// TwinCAT 3 PLC project PLC
// ProgramVersion: 3.1.4024.0
// libraries:
//   Tc2_EtherCAT, * (Beckhoff Automation GmbH)
//   Tc2_Standard, * (Beckhoff Automation GmbH)
//   Tc2_System, * (Beckhoff Automation GmbH)
//   Tc3_Module, * (Beckhoff Automation GmbH)
// project tree:
//   DUTs/ E_EP7402_CoE_Motor.TcDUT, E_EP7402_CoE_Controller.TcDUT, E_SynchronInfoData.TcDUT, ST_CoE_Parameter.TcDUT, ST_EP7402_CoE_Motor.TcDUT, ST_EP7402_CoE_Controller.TcDUT, ST_EP7402_CoE_Parameter.TcDUT, ST_EP7402_CoE_SynchronInfoData.TcDUT
//   GVLs/ GVL.TcGVL
//   / PlcTask.TcTTO
//   POUs/CoE_Access/ FB_EP7402_AutoRequestSteps.TcPOU, FB_EP7402_ReadCoEParameter.TcPOU, FB_EP7402_Scan_Motor.TcPOU, FB_EP7402_WriteCoEParameter.TcPOU
//   POUs/ MAIN.TcPOU
// real-time tasks:
//   TASK PlcTask: cycle T#2ms, priority 20, ADS port 350
// I/O:
//   DEVICE Device 3 (EtherCAT), AmsNetId 5.32.108.108.4.1
//     Box 1 (EP7402-0057) [EP7402-0057 2 Ch. BLDC Motor, 24VDC, 8x digital In/Output, B23 ENP 5G4, 1x EtherCAT junction]
// variable links:
//   PLC/PLC Instance <-> Device 3 (EtherCAT)/Box 1 (EP7402-0057)
//     PlcTask Inputs/MAIN.nEP7402Addr <-> InfoData/AdsAddr/port
//     PlcTask Inputs/MAIN.sNetId <-> InfoData/AdsAddr/netId
//     PlcTask Inputs/MAIN.stEP7402_PDOs.MDP5001_100_200_705_Input/MDP5001_100_200_705_STM_Inputs_Device_Device_Diag <-> STM Inputs Device/Device Diag
//     PlcTask Inputs/MAIN.stEP7402_PDOs.MDP5001_100_200_705_Input/MDP5001_100_DI_Inputs_Control_input_{1..4} <-> DI Inputs/Control input {1..4}  (4 links)
//     PlcTask Inputs/MAIN.stEP7402_PDOs.MDP5001_100_200_705_Input/MDP5001_100_DI_Inputs_Input_{1..4} <-> DI Inputs/Input {1..4}  (4 links)
//     PlcTask Inputs/MAIN.stEP7402_PDOs.MDP5001_100_200_705_Input/MDP5001_705_STM_Status_Channel_1_Status <-> STM Status Channel 1/Status
//     PlcTask Inputs/MAIN.stEP7402_PDOs.MDP5001_100_200_705_Input/MDP5001_705_STM_Status_Channel_2_Status <-> STM Status Channel 2/Status
//     PlcTask Inputs/MAIN.stEP7402_PDOs.MDP5001_100_200_705_Input/MDP5001_705_STM_Synchron_info_data_Channel_1_Info_data_1 <-> STM Synchron info data Channel 1/Info data 1
//     PlcTask Inputs/MAIN.stEP7402_PDOs.MDP5001_100_200_705_Input/MDP5001_705_STM_Synchron_info_data_Channel_1_Info_data_2 <-> STM Synchron info data Channel 1/Info data 2
//     PlcTask Inputs/MAIN.stEP7402_PDOs.MDP5001_100_200_705_Input/MDP5001_705_STM_Synchron_info_data_Channel_1_Info_data_3 <-> STM Synchron info data Channel 1/Info data 3
//     PlcTask Inputs/MAIN.stEP7402_PDOs.MDP5001_100_200_705_Input/MDP5001_705_STM_Synchron_info_data_Channel_2_Info_data_1 <-> STM Synchron info data Channel 2/Info data 1
//     PlcTask Inputs/MAIN.stEP7402_PDOs.MDP5001_100_200_705_Input/MDP5001_705_STM_Synchron_info_data_Channel_2_Info_data_2 <-> STM Synchron info data Channel 2/Info data 2
//     PlcTask Inputs/MAIN.stEP7402_PDOs.MDP5001_100_200_705_Input/MDP5001_705_STM_Synchron_info_data_Channel_2_Info_data_3 <-> STM Synchron info data Channel 2/Info data 3
//     PlcTask Outputs/MAIN.stEP7402_PDOs.MDP5001_100_200_705_Output/MDP5001_200_DO_Outputs_Control_output_{1..4} <-> DO Outputs/Control output {1..4}  (4 links)
//     PlcTask Outputs/MAIN.stEP7402_PDOs.MDP5001_100_200_705_Output/MDP5001_200_DO_Outputs_Output_{1..4} <-> DO Outputs/Output {1..4}  (4 links)
//     PlcTask Outputs/MAIN.stEP7402_PDOs.MDP5001_100_200_705_Output/MDP5001_705_STM_Control_Channel_1_Control <-> STM Control Channel 1/Control
//     PlcTask Outputs/MAIN.stEP7402_PDOs.MDP5001_100_200_705_Output/MDP5001_705_STM_Control_Channel_2_Control <-> STM Control Channel 2/Control
//     PlcTask Outputs/MAIN.stEP7402_PDOs.MDP5001_100_200_705_Output/MDP5001_705_STM_Target_Velocity_Channel_1_Accelleration <-> STM Target Velocity Channel 1/Accelleration
//     PlcTask Outputs/MAIN.stEP7402_PDOs.MDP5001_100_200_705_Output/MDP5001_705_STM_Target_Velocity_Channel_2_Accelleration <-> STM Target Velocity Channel 2/Accelleration
//     PlcTask Outputs/MAIN.stEP7402_PDOs.MDP5001_100_200_705_Output/MDP5001_705_STM_Target_Velocity_Channel_1_Decceleration <-> STM Target Velocity Channel 1/Decceleration
//     PlcTask Outputs/MAIN.stEP7402_PDOs.MDP5001_100_200_705_Output/MDP5001_705_STM_Target_Velocity_Channel_2_Decceleration <-> STM Target Velocity Channel 2/Decceleration
//     PlcTask Outputs/MAIN.stEP7402_PDOs.MDP5001_100_200_705_Output/MDP5001_705_STM_Target_Velocity_Channel_1_Velocity <-> STM Target Velocity Channel 1/Velocity
//     PlcTask Outputs/MAIN.stEP7402_PDOs.MDP5001_100_200_705_Output/MDP5001_705_STM_Target_Velocity_Channel_2_Velocity <-> STM Target Velocity Channel 2/Velocity

CONFIGURATION PLC
    RESOURCE PLC ON TwinCAT3
        TASK PlcTask(INTERVAL := T#2ms, PRIORITY := 20);
        PROGRAM MAIN WITH PlcTask : MAIN;
    END_RESOURCE
END_CONFIGURATION

// ---- DUTs/E_EP7402_CoE_Motor.TcDUT
{attribute 'qualified_only'}
{attribute 'strict'}
TYPE E_EP7402_CoE_Motor :
(
	Peak_Current:=1,
	Rated_Current:=2,
	Rated_Voltage:=3,
	Phase_To_Phase_Resistance:=4,
	Start_Velocity:=5,
	Mechanical_To_Electrical_Ratio:=6,
	Rated_Velocity:=7,
	I2T_Warn_Level:=8,
	I2T_Error_Level:=9,
	Motor_Thermal_Time_Constant:=10
);
END_TYPE

// ---- DUTs/E_EP7402_CoE_Controller.TcDUT
{attribute 'qualified_only'}
{attribute 'strict'}
TYPE E_EP7402_CoE_Controller :
(
	Disable_Motor_Diagnosis:=1,
	Disable_I2T_Current_Limiting:=2,
	Velocity_Loop_Integral_Time:=3,
	Velocity_Loop_Proportional_Gain:=4,
	Velocity_Feed_Forward_Gain:=5,
	Sensorless_Offset_Scaling:=6,
	Align_Duration:=7,
	Rampup_Duration:=8,
	Rampup_Velocity:=9,	
	Rampup_Needed_Switchover_Events:=10,
	Commutation_Threshold:=11,
	Current_Loop_Proportional_Gain:=12,
	Current_Loop_Integral_Time:=13,
	Restart_After_Error_Number_Of_Repetition:=14,
	Restart_After_Error_Delay:=15
);
END_TYPE

// ---- DUTs/E_SynchronInfoData.TcDUT
{attribute 'qualified_only'}
TYPE E_SynchronInfoData :
(
	Motor_velocity 				:= 7,
	Motor_velocity_filtered 	:= 8,
	Motor_I2T_load 				:= 11,
	Amplifier_I2T_load 			:= 12,
	Motor_dc_current 			:= 13,
	Motor_dc_current_filtered 	:= 14,
	Motor_back_emf 				:= 17,
	Motor_restart_counter 		:= 18,
	Internal_temperature 		:= 101,
	Motor_supply_voltage 		:= 104,
	none
)USINT:=none;
END_TYPE

// ---- DUTs/ST_CoE_Parameter.TcDUT
TYPE ST_CoE_Parameter :
STRUCT
	sSubIndex		: STRING;	// Number of Index:Subindex
	sDescription	: STRING;	// Description of CoE Parameter
	nValue			: UDINT;	// Set Value to change CoE Parameter 
	nReadValue		: UDINT;	// Actual Value of Parameterread from terminal
	sValueRange		: STRING;	// Description of the range of the parameter 
END_STRUCT
END_TYPE

// ---- DUTs/ST_EP7402_CoE_Motor.TcDUT
 {attribute 'pack_mode' := '0'}
 // Represents data struct of COE Index 8020/8030 --> can be determined in esi
TYPE ST_EP7402_CoE_Motor :
STRUCT
	Sub_Index_res_0: ARRAY [1..2] OF BYTE;
	Sub_Index_001: UINT;
	Sub_Index_002: UINT;
	Sub_Index_003: UINT;
	Sub_Index_004: UINT;
	Sub_Index_res_1: ARRAY [1..8] OF BYTE;
	Sub_Index_009: UINT;
	Sub_Index_res_2: ARRAY [1..8] OF BYTE;	
	Sub_Index_019: UINT;
	Sub_Index_020: UINT;
	Sub_Index_res_3: ARRAY [1..2] OF BYTE;	
	Sub_Index_022: USINT;
	Sub_Index_024: USINT;
	Sub_Index_025: UINT;
	Sub_Index_res_4: ARRAY [1..2] OF BYTE;	
END_STRUCT
END_TYPE

// ---- DUTs/ST_EP7402_CoE_Controller.TcDUT
 {attribute 'pack_mode' := '0'}
 // Represents data struct of COE Index 8023/8033 --> can be determined in esi
TYPE ST_EP7402_CoE_Controller :
STRUCT
	Bit_Reserved_001 :BIT;
	Bit_Reserved_002 :BIT;
	Bit_Reserved_003 :BIT;
	Bit_Reserved_004 :BIT;
	Bit_Reserved_005 :BIT;
	Bit_Reserved_006 :BIT;
	Bit_Reserved_007 :BIT;
	Bit_Reserved_008 :BIT;
	Bit_Reserved_009 :BIT;
	Bit_Reserved_010 :BIT;
	Bit_Reserved_011 :BIT;
	Bit_Reserved_012 :BIT;
	Bit_Reserved_013 :BIT;
	Bit_Reserved_014 :BIT;
	Bit_Reserved_015 :BIT;
	Bit_Reserved_016 :BIT;
	Bit_Reserved_017 :BIT;
	Sub_Index_002: BIT;
	Sub_Index_003: BIT;
	Sub_Index_004: BIT;
	Bit_Reserved_021 :BIT;
	Bit_Reserved_022 :BIT;
	Bit_Reserved_023 :BIT;
	Bit_Reserved_024 :BIT;
	Bit_Reserved_025 :BIT;
	Bit_Reserved_026 :BIT;
	Bit_Reserved_027 :BIT;
	Bit_Reserved_028 :BIT;
	Bit_Reserved_029 :BIT;
	Bit_Reserved_030 :BIT;
	Bit_Reserved_031 :BIT;
	Bit_Reserved_032 :BIT;
	Sub_Index_017: UDINT;
	Sub_Index_018: UDINT;
	Sub_Index_019: USINT;
	Sub_Index_020: SINT;
	Sub_Index_021: UINT;
	Byte_Reserved_001 :ARRAY[1..2] OF BYTE;
	Sub_Index_024: UINT;
	Sub_Index_025: UINT;
	Sub_Index_033: UINT;
	Sub_Index_034: UINT;
	Sub_Index_035: UINT;
	Sub_Index_036: UINT;
	Sub_Index_037: UINT;
	Sub_Index_038: UINT;
END_STRUCT
END_TYPE

// ---- DUTs/ST_EP7402_CoE_Parameter.TcDUT
TYPE ST_EP7402_CoE_Parameter :
STRUCT
	astCoE_Parameter_Motor				: ARRAY[1..2] OF ARRAY [1..gvl.cnNumberOfCoeParameter_Motor] OF ST_CoE_Parameter :=
	[[
		(sSubIndex:='8020:01',	sDescription:='Peak current[mA]'					,nValue:=0,nReadValue:=0, sValueRange:='<5000'),
		(sSubIndex:='8020:02',	sDescription:='Rated current[mA]'					,nValue:=0,nReadValue:=0, sValueRange:='<3500'),
		(sSubIndex:='8020:03',	sDescription:='Rated Voltage [0.01 V]'				,nValue:=0,nReadValue:=0, sValueRange:='<2400'),
		(sSubIndex:='8020:04',	sDescription:='Phase to phase resistance [0.01 Ω]'	,nValue:=0,nReadValue:=0, sValueRange:='-'),
		(sSubIndex:='8020:09',	sDescription:='Start velocity [°/s]'				,nValue:=0,nReadValue:=0, sValueRange:='-'),
		(sSubIndex:='8020:13',	sDescription:='Mechanical to electrical ratio'		,nValue:=0,nReadValue:=0, sValueRange:='-'),
		(sSubIndex:='8020:14',	sDescription:='Rated velocity [°/s]'				,nValue:=0,nReadValue:=0, sValueRange:='-'),
		(sSubIndex:='8020:16',	sDescription:='I2T warn level [%]'					,nValue:=0,nReadValue:=0, sValueRange:='-'),
		(sSubIndex:='8020:18',	sDescription:='I2T error level [%]'					,nValue:=0,nReadValue:=0, sValueRange:='-'),
		(sSubIndex:='8020:19',	sDescription:='Motor thermal time constant [0.1s]'	,nValue:=0,nReadValue:=0, sValueRange:='-')
	],
	[
		(sSubIndex:='8030:01',	sDescription:='Peak current[mA]'					,nValue:=0,nReadValue:=0, sValueRange:='<5000'),
		(sSubIndex:='8030:02',	sDescription:='Rated current[mA]'					,nValue:=0,nReadValue:=0, sValueRange:='<3500'),
		(sSubIndex:='8030:03',	sDescription:='Rated Voltage [0.01 V]'				,nValue:=0,nReadValue:=0, sValueRange:='<2400'),
		(sSubIndex:='8030:04',	sDescription:='Phase to phase resistance [0.01 Ω]'	,nValue:=0,nReadValue:=0, sValueRange:='-'),
		(sSubIndex:='8030:09',	sDescription:='Start velocity [°/s]'				,nValue:=0,nReadValue:=0, sValueRange:='-'),
		(sSubIndex:='8030:13',	sDescription:='Mechanical to electrical ratio'		,nValue:=0,nReadValue:=0, sValueRange:='-'),
		(sSubIndex:='8030:14',	sDescription:='Rated velocity [°/s]'				,nValue:=0,nReadValue:=0, sValueRange:='-'),
		(sSubIndex:='8030:16',	sDescription:='I2T warn level [%]'					,nValue:=0,nReadValue:=0, sValueRange:='-'),
		(sSubIndex:='8030:18',	sDescription:='I2T error level [%]'					,nValue:=0,nReadValue:=0, sValueRange:='-'),
		(sSubIndex:='8030:19',	sDescription:='Motor thermal time constant [0.1s]'	,nValue:=0,nReadValue:=0, sValueRange:='-')
	]];
	
	astCoE_Parameter_Controller			: ARRAY[1..2] OF ARRAY [1..gvl.cnNumberOfCoeParameter_Controller] OF ST_CoE_Parameter :=
		[[
			(sSubIndex:='8023:03',	sDescription:='Disable motor diagnosis'						,nValue:=0,nReadValue:=0, sValueRange:='0/1'),
			(sSubIndex:='8023:04',	sDescription:='Disable I2T current limiting'				,nValue:=0,nReadValue:=0, sValueRange:='0/1'),
			(sSubIndex:='8023:11',	sDescription:='Velocity loop integral time [0.1ms]'			,nValue:=0,nReadValue:=0, sValueRange:='-'),
            (sSubIndex:='8023:12',	sDescription:='Velocity loop proportional gain [uV/(°/s)]'	,nValue:=0,nReadValue:=0, sValueRange:='-'),
            (sSubIndex:='8023:13',	sDescription:='Velocity feed forward'						,nValue:=0,nReadValue:=0, sValueRange:='-'),
            (sSubIndex:='8023:14',	sDescription:='Sensorless offset scaling {%]'				,nValue:=0,nReadValue:=0, sValueRange:='-'),
            (sSubIndex:='8023:15',	sDescription:='Align duration [ms]'							,nValue:=0,nReadValue:=0, sValueRange:='-'),
            (sSubIndex:='8023:18',	sDescription:='Rampup duration [ms]'						,nValue:=0,nReadValue:=0, sValueRange:='-'),
            (sSubIndex:='8023:19',	sDescription:='Rampup velocity [°/s]'						,nValue:=0,nReadValue:=0, sValueRange:='-'),
            (sSubIndex:='8023:21',	sDescription:='Rampup needed switchover events'				,nValue:=0,nReadValue:=0, sValueRange:='-'),
            (sSubIndex:='8023:22',	sDescription:='Commutation Threshold'						,nValue:=0,nReadValue:=0, sValueRange:='-'),
            (sSubIndex:='8023:23',	sDescription:='Current loop proportional gain [0.1V/A]'		,nValue:=0,nReadValue:=0, sValueRange:='-'),
            (sSubIndex:='8023:24',	sDescription:='Current Loop integral time [0.1ms]'			,nValue:=0,nReadValue:=0, sValueRange:='-'),
            (sSubIndex:='8023:25',	sDescription:='Restart after error number of repetition'	,nValue:=0,nReadValue:=0, sValueRange:='-'),
            (sSubIndex:='8023:26',	sDescription:='Restart after error delay [ms]'					,nValue:=0,nReadValue:=0, sValueRange:='-')
		],
		[
			(sSubIndex:='8033:03',	sDescription:='Disable motor diagnosis'						,nValue:=0,nReadValue:=0, sValueRange:='0/1'),
			(sSubIndex:='8033:04',	sDescription:='Disable I2T current limiting'				,nValue:=0,nReadValue:=0, sValueRange:='0/1'),
			(sSubIndex:='8033:11',	sDescription:='Velocity loop integral time [0.1ms]'			,nValue:=0,nReadValue:=0, sValueRange:='-'),
            (sSubIndex:='8033:12',	sDescription:='Velocity loop proportional gain [uV/(°/s)]'	,nValue:=0,nReadValue:=0, sValueRange:='-'),
            (sSubIndex:='8033:13',	sDescription:='Velocity feed forward'						,nValue:=0,nReadValue:=0, sValueRange:='-'),
            (sSubIndex:='8033:14',	sDescription:='Sensorless offset scaling {%]'				,nValue:=0,nReadValue:=0, sValueRange:='-'),
            (sSubIndex:='8033:15',	sDescription:='Align duration [ms]'							,nValue:=0,nReadValue:=0, sValueRange:='-'),
            (sSubIndex:='8033:18',	sDescription:='Rampup duration [ms]'						,nValue:=0,nReadValue:=0, sValueRange:='-'),
            (sSubIndex:='8033:19',	sDescription:='Rampup velocity [°/s]'						,nValue:=0,nReadValue:=0, sValueRange:='-'),
            (sSubIndex:='8033:21',	sDescription:='Rampup needed switchover events'				,nValue:=0,nReadValue:=0, sValueRange:='-'),
            (sSubIndex:='8033:22',	sDescription:='Commutation Threshold'						,nValue:=0,nReadValue:=0, sValueRange:='-'),
            (sSubIndex:='8033:23',	sDescription:='Current loop proportional gain [0.1V/A]'		,nValue:=0,nReadValue:=0, sValueRange:='-'),
            (sSubIndex:='8033:24',	sDescription:='Current Loop integral time [0.1ms]'		   	,nValue:=0,nReadValue:=0, sValueRange:='-'),
            (sSubIndex:='8033:25',	sDescription:='Restart after error number of repetition'	,nValue:=0,nReadValue:=0, sValueRange:='-'),
            (sSubIndex:='8033:26',	sDescription:='Restart after error delay [ms]'				,nValue:=0,nReadValue:=0, sValueRange:='-')
		]];
		astCoE_Parameter_SynchronInfoData	: ARRAY [1..2] OF ARRAY [1..3] OF E_SynchronInfoData;
END_STRUCT 
END_TYPE

// ---- DUTs/ST_EP7402_CoE_SynchronInfoData.TcDUT
 {attribute 'pack_mode' := '0'}
// Represents data struct of COE Index 8022/8032 --> can be determined in esi
TYPE ST_EP7402_CoE_SynchronInfoData :
STRUCT
	aSub_Index_res_000 : ARRAY [1..4] OF BYTE;
	nInfoData1 : USINT;
	nInfoData2 : USINT;
	aSub_Index_res_001 : ARRAY [1..6] OF BYTE;
	nInfoData3 : USINT;
	aSub_Index_res_002 : ARRAY [1..3] OF BYTE;	
END_STRUCT
END_TYPE

// ---- GVLs/GVL.TcGVL
{attribute 'qualified_only'}
VAR_GLOBAL CONSTANT
	cnNumberOfCoeParameter_Motor:USINT:=10;
	cnNumberOfCoeParameter_Controller:USINT:=15;
	cnSubIndex_ResetDeliveryStatus: BYTE:=16#1;
	cnIndex_ResetDeliveryStatus: WORD:=16#1011;
	cnResetParameter : UDINT:= 1684107116;
END_VAR

// ---- POUs/MAIN.TcPOU
PROGRAM MAIN
VAR
	// Variables to link with HW
	sNetId			AT%I*	: T_AmsNetIdArr;				// link with PDO: EP7402 -->InfoData --> AdsAddr.netId
	nEP7402Addr		AT%I*	: UINT := 1001;					// link with PDO: EP7402 -->InfoData --> AdsAddr.port
	stEP7402_PDOs			: MDP5001_100_200_705_F94A9C2E;	// Struct for simple Link with Box: EP7402 --> PLC --> Create PLC Data Type --> disable "Per Channel"
															// --> Link To PLC.. --> Select Struct this struct

	// Function blocks used for COE access 
	fbEP7402_ReadCoE 			: FB_EP7402_ReadCoEParameter; 	// Read Coe Settings for Motor Configuration: Index 8020/30 and 8023/33 of a box
	fbEP7402_WriteCoE 			: FB_EP7402_WriteCoEParameter;	// Write Coe Settings for Motor Configuration: Index 8020/30 and 8023/33 of a box
	fbEP7402_AutoRequestSteps	: FB_EP7402_AutoRequestSteps;	// Sending Request for single Motor steps. Needed to determine "Mechanical to electrical Ratio"
	fbEP7402_ScanMotor			: FB_EP7402_Scan_Motor;			// Sending Request to start Motor Scan. Needed to determine controller values.
	fbResetCoE_Parameter 		: FB_EcCoESdoWrite;				// Reset Box --> reset to delivery status
	
	// structs storing CoE-Parameters
	stLast_EP7402_CoE_Parameter : ST_EP7402_CoE_Parameter;		// Struct with Coe Paramters in last PLC Cycle --> needed for getting changes
	st_EP7402_CoE_Parameter 	: ST_EP7402_CoE_Parameter;		// Struct containing all current CoE Data (also inputs from HMI)
	
	fbCoeWriteFinished			: f_trig;
	fbReadFinished				: f_trig;
	bReadCoE					: BOOL;
	bMotorChannel_1_Selected	: BOOL:=True;
	nIndex						: UINT;	
	nResetParameter 			: UDINT;
	bInit						: BOOL;
END_VAR

GetEvents();
Init();

// Reset Box to delivery state (can be triggered from HMI)
fbResetCoE_Parameter(	sNetID:=F_CreateAmsNetId(sNetId),
						nSlaveAddr:=nEP7402Addr, 
						nSubIndex := gvl.cnSubIndex_ResetDeliveryStatus, 
						nIndex := gvl.cnIndex_ResetDeliveryStatus,	
						pSrcBuf := ADR(gvl.cnResetParameter),
						cbBufLen := SIZEOF(gvl.cnResetParameter),
						bExecute := fbResetCoE_Parameter.bExecute
						);

// special configuration functions requested via CoE (can be triggered from HMI)
	//Request single Motor Steps
	fbEP7402_AutoRequestSteps(bEnable:=fbEP7402_AutoRequestSteps.bEnable, bMotorChannel_1:=bMotorChannel_1_Selected,sNetID:=F_CreateAmsNetId(sNetId),nSlaveAddr:=nEP7402Addr);
	//Request Motor Scan
	fbEP7402_ScanMotor(bExecute:=fbEP7402_ScanMotor.bExecute, bMotorChannel_1:=bMotorChannel_1_Selected,sNetID:=F_CreateAmsNetId(sNetId),nSlaveAddr:=nEP7402Addr);

ACTION GetEvents:


// A Coe Write has finished --> Read is necessary
fbCoeWriteFinished(clk:=fbEP7402_WriteCoE.bBusy OR fbResetCoE_Parameter.bBusy OR fbEP7402_ScanMotor.bBusy);

// Read in CoE Parameters of Box
fbEP7402_ReadCoE(bExecute:=fbCoeWriteFinished.q OR fbEP7402_ReadCoE.bExecute AND NOT fbEP7402_WriteCoE.bBusy , stEP7402_CoE_Parameter  :=st_EP7402_CoE_Parameter);
// A Coe Read is finished
fbReadFinished(clk:=fbEP7402_ReadCoE.bBusy );
IF fbReadFinished.Q THEN
	fbEP7402_ReadCoE.bExecute:=false;
	initCoEValues();
END_IF

// Write Coe Parameters if set parameters have been changed (HMI)
fbEP7402_WriteCoE(bExecute:=FALSE, stEP7402_CoE_Parameter  :=st_EP7402_CoE_Parameter);
IF memcmp(ADR(stLast_EP7402_CoE_Parameter),ADR(st_EP7402_CoE_Parameter),SIZEOF(st_EP7402_CoE_Parameter))<>0 AND NOT fbEP7402_ReadCoE.bBusy THEN 
	fbEP7402_WriteCoE(bExecute:=TRUE, sNetID:=F_CreateAmsNetId(sNetId),nSlaveAddr:=nEP7402Addr, stEP7402_CoE_Parameter  :=st_EP7402_CoE_Parameter);
	stLast_EP7402_CoE_Parameter:=st_EP7402_CoE_Parameter;
END_IF
END_ACTION

ACTION Init:
IF NOT bInit THEN
	fbEP7402_ReadCoE(bExecute:=NOT fbEP7402_ReadCoE.bBusy,sNetID:=F_CreateAmsNetId(sNetId),nSlaveAddr:=nEP7402Addr, stEP7402_CoE_Parameter  :=st_EP7402_CoE_Parameter);
	IF NOT fbEP7402_ReadCoE.bBusy THEN
		bInit:=TRUE;
		initCoEValues();
	END_IF
END_IF
END_ACTION

ACTION InitCoEValues:
FOR nIndex:= 1 TO gvl.cnNumberOfCoeParameter_Motor DO
	st_EP7402_CoE_Parameter.astCoE_Parameter_Motor[1][nIndex].nValue:=st_EP7402_CoE_Parameter.astCoE_Parameter_Motor[1][nIndex].nReadValue;
	st_EP7402_CoE_Parameter.astCoE_Parameter_Motor[2][nIndex].nValue:=st_EP7402_CoE_Parameter.astCoE_Parameter_Motor[2][nIndex].nReadValue;
END_FOR
FOR nIndex:= 1 TO gvl.cnNumberOfCoeParameter_Controller DO
	st_EP7402_CoE_Parameter.astCoE_Parameter_Controller[1][nIndex].nValue:=st_EP7402_CoE_Parameter.astCoE_Parameter_Controller[1][nIndex].nReadValue;
	st_EP7402_CoE_Parameter.astCoE_Parameter_Controller[2][nIndex].nValue:=st_EP7402_CoE_Parameter.astCoE_Parameter_Controller[2][nIndex].nReadValue;
END_FOR
stLast_EP7402_CoE_Parameter:=st_EP7402_CoE_Parameter;
END_ACTION

END_PROGRAM

// ---- POUs/CoE_Access/FB_EP7402_ReadCoEParameter.TcPOU

FUNCTION_BLOCK FB_EP7402_ReadCoEParameter
VAR_IN_OUT 
	stEP7402_CoE_Parameter	: ST_EP7402_CoE_Parameter;		
END_VAR
VAR_INPUT
	bExecute	: BOOL;
	sNetId 		: T_AmsNetID;
	nSlaveAddr	: UINT;
END_VAR
VAR_OUTPUT
	bBusy:BOOL;
	bError:BOOL;
	nErrId:UDINT;
END_VAR
VAR
	fbReadCoEParameterEx				:  FB_EcCoESdoReadEx;
	nParameter							:  UINT;
	nStep								: (init, StartRead_MotorParameter_1, Reading_MotorParameter_1, StartRead_ControllerParameter_1, Reading_ControllerParameter_1, StartRead_SynchronInfoData_1, Reading_SynchronInfoData_1,
											StartRead_MotorParameter_2, Reading_MotorParameter_2, StartRead_ControllerParameter_2, Reading_ControllerParameter_2, StartRead_SynchronInfoData_2, Reading_SynchronInfoData_2);
	stCoe_Read_Motor					: ST_EP7402_CoE_Motor;
	stCoe_Read_Controller				: ST_EP7402_CoE_Controller;
	stCoe_Read_SynchronInfoData			: ST_EP7402_CoE_SynchronInfoData;
	fbExecuteTrigger				 	: r_trig;
	nIndex: uint;
END_VAR

fbExecuteTrigger(clk:=bExecute);
IF fbExecuteTrigger.q THEN
	nStep:=StartRead_MotorParameter_1;
	bBusy:=TRUE;
END_IF

CASE nStep OF
	init:
		bBusy := FALSE;
		bError:=fbReadCoEParameterEx.bError;
		nErrId:=fbReadCoEParameterEx.nErrId;
	
	StartRead_MotorParameter_1:
		fbReadCoEParameterEx(bExecute:=FALSE);
		IF NOT fbReadCoEParameterEx.bBusy THEN
			fbReadCoEParameterEx(
				sNetId:= sNetId, 
				nSlaveAddr:= nSlaveAddr, 
				nIndex:= 16#8020, 
				pDstBuf:= ADR(stCoe_Read_Motor), 
				cbBufLen:= SIZEOF(stCoe_Read_Motor), 
				bExecute:= TRUE,
				bCompleteAccess:= TRUE);
			nStep:=	Reading_MotorParameter_1;
		END_IF

		
	Reading_MotorParameter_1:
		fbReadCoEParameterEx(bExecute:=FALSE);
		IF NOT fbReadCoEParameterEx.bBusy THEN
			IF fbReadCoEParameterEx.bError THEN
				nStep:= init;
			ELSE
				TransferBufferDataToStruct_Motor(nChannel:=1);
				nStep:= StartRead_ControllerParameter_1;
			END_IF
		END_IF
	
	StartRead_ControllerParameter_1:
		fbReadCoEParameterEx(bExecute:=FALSE);
		IF NOT fbReadCoEParameterEx.bBusy THEN
			fbReadCoEParameterEx(
				sNetId:= sNetId, 
				nSlaveAddr:= nSlaveAddr, 
				nIndex:= 16#8023, 
				pDstBuf:= ADR(stCoe_Read_Controller), 
				cbBufLen:= SIZEOF(stCoe_Read_Controller), 
				bExecute:= TRUE,
				bCompleteAccess:= TRUE);
			nStep:=	Reading_ControllerParameter_1;
		END_IF
		
	Reading_ControllerParameter_1:
		fbReadCoEParameterEx(bExecute:=FALSE);
		IF NOT fbReadCoEParameterEx.bBusy THEN
			IF fbReadCoEParameterEx.bError THEN
				nStep:= init;
			ELSE
				TransferBufferDataToStruct_Controller(nChannel:=1);
				nStep:= StartRead_SynchronInfoData_1;
			END_IF
		END_IF
		
	StartRead_SynchronInfoData_1:
		fbReadCoEParameterEx(bExecute:=FALSE);
			IF NOT fbReadCoEParameterEx.bBusy THEN
				fbReadCoEParameterEx(
					sNetId:= sNetId, 
					nSlaveAddr:= nSlaveAddr, 
					nIndex:= 16#8022, 
					pDstBuf:= ADR(stCoe_Read_SynchronInfoData), 
					cbBufLen:= SIZEOF(stCoe_Read_SynchronInfoData), 
					bExecute:= TRUE,
					bCompleteAccess:= TRUE);
				nStep:=	Reading_SynchronInfoData_1;
			END_IF
	
	Reading_SynchronInfoData_1:
		fbReadCoEParameterEx(bExecute:=FALSE);
			IF NOT fbReadCoEParameterEx.bBusy THEN
				IF fbReadCoEParameterEx.bError THEN
					nStep:= init;
				ELSE
					TransferBufferDataToStruct_SynchronInfoData(nChannel:=1);
					nStep:= StartRead_MotorParameter_2;
				END_IF
			END_IF
		
	StartRead_MotorParameter_2:
		fbReadCoEParameterEx(bExecute:=FALSE);
		IF NOT fbReadCoEParameterEx.bBusy THEN
			fbReadCoEParameterEx(
				sNetId:= sNetId, 
				nSlaveAddr:= nSlaveAddr, 
				nIndex:= 16#8030, 
				pDstBuf:= ADR(stCoe_Read_Motor), 
				cbBufLen:= SIZEOF(stCoe_Read_Motor), 
				bExecute:= TRUE,
				bCompleteAccess:= TRUE);
			nStep:=	Reading_MotorParameter_2;
		END_IF

		
	Reading_MotorParameter_2:
		fbReadCoEParameterEx(bExecute:=FALSE);
		IF NOT fbReadCoEParameterEx.bBusy THEN
			IF fbReadCoEParameterEx.bError THEN
				nStep:= init;
			ELSE
				TransferBufferDataToStruct_Motor(nChannel:=2);
				nStep:= StartRead_ControllerParameter_2;
			END_IF
		END_IF
	
	StartRead_ControllerParameter_2:
		fbReadCoEParameterEx(bExecute:=FALSE);
		IF NOT fbReadCoEParameterEx.bBusy THEN
			fbReadCoEParameterEx(
				sNetId:= sNetId, 
				nSlaveAddr:= nSlaveAddr, 
				nIndex:= 16#8033, 
				pDstBuf:= ADR(stCoe_Read_Controller), 
				cbBufLen:= SIZEOF(stCoe_Read_Controller), 
				bExecute:= TRUE,
				bCompleteAccess:= TRUE);
			nStep:=	Reading_ControllerParameter_2;
		END_IF
		
	Reading_ControllerParameter_2:
		fbReadCoEParameterEx(bExecute:=FALSE);
		IF NOT fbReadCoEParameterEx.bBusy THEN
			IF fbReadCoEParameterEx.bError THEN
				nStep:= init;
			ELSE 
				TransferBufferDataToStruct_Controller(nChannel:=2);
				nStep:= StartRead_SynchronInfoData_2;
			END_IF
		END_IF
		
	StartRead_SynchronInfoData_2:
		fbReadCoEParameterEx(bExecute:=FALSE);
		IF NOT fbReadCoEParameterEx.bBusy THEN
			fbReadCoEParameterEx(
				sNetId:= sNetId, 
				nSlaveAddr:= nSlaveAddr, 
				nIndex:= 16#8032, 
				pDstBuf:= ADR(stCoe_Read_SynchronInfoData), 
				cbBufLen:= SIZEOF(stCoe_Read_SynchronInfoData), 
				bExecute:= TRUE,
				bCompleteAccess:= TRUE);
			nStep:=	Reading_SynchronInfoData_2;
		END_IF
		
	Reading_SynchronInfoData_2:
		fbReadCoEParameterEx(bExecute:=FALSE);
		IF NOT fbReadCoEParameterEx.bBusy THEN
			IF NOT fbReadCoEParameterEx.bError THEN
				TransferBufferDataToStruct_SynchronInfoData(nChannel:=2);
			END_IF
			nStep:= init;
		END_IF
		
END_CASE

METHOD TransferBufferDataToStruct_Controller
VAR_INPUT
	nChannel:USINT;
END_VAR
// The warning can be disabled here as the user is aware of the risk that the reference may not be valid by checking its validity
{warning disable C0371}

IF nChannel=1 OR nChannel=2  AND __ISVALIDREF(stEP7402_CoE_Parameter)THEN
	stEP7402_CoE_Parameter.astCoE_Parameter_Controller[nChannel][E_EP7402_CoE_Controller.Disable_Motor_Diagnosis].nReadValue:=TO_UDINT(stCoe_Read_Controller.Sub_Index_003);
	stEP7402_CoE_Parameter.astCoE_Parameter_Controller[nChannel][E_EP7402_CoE_Controller.Disable_I2T_Current_Limiting].nReadValue:=TO_UDINT(stCoe_Read_Controller.Sub_Index_004);
	stEP7402_CoE_Parameter.astCoE_Parameter_Controller[nChannel][E_EP7402_CoE_Controller.Velocity_Loop_Integral_Time].nReadValue:=TO_UDINT(stCoe_Read_Controller.Sub_Index_017);
	stEP7402_CoE_Parameter.astCoE_Parameter_Controller[nChannel][E_EP7402_CoE_Controller.Velocity_Loop_Proportional_Gain].nReadValue:=TO_UDINT(stCoe_Read_Controller.Sub_Index_018);
	stEP7402_CoE_Parameter.astCoE_Parameter_Controller[nChannel][E_EP7402_CoE_Controller.Velocity_Feed_Forward_Gain].nReadValue:=TO_UDINT(stCoe_Read_Controller.Sub_Index_019);
	stEP7402_CoE_Parameter.astCoE_Parameter_Controller[nChannel][E_EP7402_CoE_Controller.Sensorless_Offset_Scaling].nReadValue:=TO_UDINT(stCoe_Read_Controller.Sub_Index_020);
	stEP7402_CoE_Parameter.astCoE_Parameter_Controller[nChannel][E_EP7402_CoE_Controller.Align_Duration].nReadValue:=TO_UDINT(stCoe_Read_Controller.Sub_Index_021);
	stEP7402_CoE_Parameter.astCoE_Parameter_Controller[nChannel][E_EP7402_CoE_Controller.Rampup_Duration].nReadValue:=TO_UDINT(stCoe_Read_Controller.Sub_Index_024);
	stEP7402_CoE_Parameter.astCoE_Parameter_Controller[nChannel][E_EP7402_CoE_Controller.Rampup_Velocity].nReadValue:=TO_UDINT(stCoe_Read_Controller.Sub_Index_025);
	stEP7402_CoE_Parameter.astCoE_Parameter_Controller[nChannel][E_EP7402_CoE_Controller.Rampup_Needed_Switchover_Events].nReadValue:=TO_UDINT(stCoe_Read_Controller.Sub_Index_033);
	stEP7402_CoE_Parameter.astCoE_Parameter_Controller[nChannel][E_EP7402_CoE_Controller.Commutation_Threshold].nReadValue:=TO_UDINT(stCoe_Read_Controller.Sub_Index_034);
	stEP7402_CoE_Parameter.astCoE_Parameter_Controller[nChannel][E_EP7402_CoE_Controller.Current_Loop_Proportional_Gain].nReadValue:=TO_UDINT(stCoe_Read_Controller.Sub_Index_035);
	stEP7402_CoE_Parameter.astCoE_Parameter_Controller[nChannel][E_EP7402_CoE_Controller.Current_Loop_Integral_Time].nReadValue:=TO_UDINT(stCoe_Read_Controller.Sub_Index_036);
	stEP7402_CoE_Parameter.astCoE_Parameter_Controller[nChannel][E_EP7402_CoE_Controller.Restart_After_Error_Number_Of_Repetition].nReadValue:=TO_UDINT(stCoe_Read_Controller.Sub_Index_037);
	stEP7402_CoE_Parameter.astCoE_Parameter_Controller[nChannel][E_EP7402_CoE_Controller.Restart_After_Error_Delay].nReadValue:=TO_UDINT(stCoe_Read_Controller.Sub_Index_038);
END_IF
END_METHOD

METHOD TransferBufferDataToStruct_Motor
VAR_INPUT
	nChannel:USINT;
END_VAR
// The warning can be disabled here as the user is aware of the risk that the reference may not be valid by checking its validity
{warning disable C0371}

IF nChannel=1 OR nChannel=2 and __ISVALIDREF(stEP7402_CoE_Parameter) THEN
	stEP7402_CoE_Parameter.astCoE_Parameter_Motor[nChannel][E_EP7402_CoE_Motor.Peak_Current].nReadValue:=stCoe_Read_Motor.Sub_Index_001;
	stEP7402_CoE_Parameter.astCoE_Parameter_Motor[nChannel][E_EP7402_CoE_Motor.Rated_Current].nReadValue:=stCoe_Read_Motor.Sub_Index_002;
	stEP7402_CoE_Parameter.astCoE_Parameter_Motor[nChannel][E_EP7402_CoE_Motor.Rated_Voltage].nReadValue:=stCoe_Read_Motor.Sub_Index_003;
	stEP7402_CoE_Parameter.astCoE_Parameter_Motor[nChannel][E_EP7402_CoE_Motor.Phase_To_Phase_Resistance].nReadValue:=stCoe_Read_Motor.Sub_Index_004;
	stEP7402_CoE_Parameter.astCoE_Parameter_Motor[nChannel][E_EP7402_CoE_Motor.Start_Velocity].nReadValue:=stCoe_Read_Motor.Sub_Index_009;
	stEP7402_CoE_Parameter.astCoE_Parameter_Motor[nChannel][E_EP7402_CoE_Motor.Mechanical_To_Electrical_Ratio].nReadValue:=stCoe_Read_Motor.Sub_Index_019;
	stEP7402_CoE_Parameter.astCoE_Parameter_Motor[nChannel][E_EP7402_CoE_Motor.Rated_Velocity].nReadValue:=stCoe_Read_Motor.Sub_Index_020;
	stEP7402_CoE_Parameter.astCoE_Parameter_Motor[nChannel][E_EP7402_CoE_Motor.I2T_Warn_Level].nReadValue:=stCoe_Read_Motor.Sub_Index_022;
	stEP7402_CoE_Parameter.astCoE_Parameter_Motor[nChannel][E_EP7402_CoE_Motor.I2T_Error_Level].nReadValue:=stCoe_Read_Motor.Sub_Index_024;
	stEP7402_CoE_Parameter.astCoE_Parameter_Motor[nChannel][E_EP7402_CoE_Motor.Motor_Thermal_Time_Constant].nReadValue:=stCoe_Read_Motor.Sub_Index_025;
END_IF
END_METHOD

METHOD TransferBufferDataToStruct_SynchronInfoData
VAR_INPUT
	nChannel:USINT;
END_VAR
// The warning can be disabled here as the user is aware of the risk that the reference may not be valid by checking its validity
{warning disable C0371}

IF nChannel=1 OR nChannel=2 and __ISVALIDREF(stEP7402_CoE_Parameter) THEN
	stEP7402_CoE_Parameter.astCoE_Parameter_SynchronInfoData[nChannel][1]:=stCoe_Read_SynchronInfoData.nInfoData1;
	stEP7402_CoE_Parameter.astCoE_Parameter_SynchronInfoData[nChannel][2]:=stCoe_Read_SynchronInfoData.nInfoData2;
	stEP7402_CoE_Parameter.astCoE_Parameter_SynchronInfoData[nChannel][3]:=stCoe_Read_SynchronInfoData.nInfoData3;
END_IF
END_METHOD

END_FUNCTION_BLOCK

// ---- POUs/CoE_Access/FB_EP7402_WriteCoEParameter.TcPOU
FUNCTION_BLOCK FB_EP7402_WriteCoEParameter
VAR_IN_OUT 
	stEP7402_CoE_Parameter	: ST_EP7402_CoE_Parameter;		
END_VAR
VAR_INPUT
	bExecute	: BOOL;
	sNetId 		: T_AmsNetID;
	nSlaveAddr	: UINT;
END_VAR
VAR_OUTPUT
	bBusy:BOOL;
	bError:BOOL;
	nErrId:UDINT;
END_VAR
VAR
	fbWriteCoEParameterEx				:  FB_EcCoESdoWriteEx;
	nParameter							:  UINT;
	nStep								: (init, StartSend_MotorParameter_1, Sending_MotorParameter_1, StartSend_ControllerParameter_1, Sending_ControllerParameter_1, StartSend_SynchronInfoData_1, Sending_SynchronInfoData_1,
											StartSend_MotorParameter_2, Sending_MotorParameter_2, StartSend_ControllerParameter_2, Sending_ControllerParameter_2, StartSend_SynchronInfoData_2, Sending_SynchronInfoData_2);
	stCoe_Write_Motor					: ST_EP7402_CoE_Motor;
	stCoe_Write_Controller				: ST_EP7402_CoE_Controller;
	stCoe_Write_SynchronInfoData		: ST_EP7402_CoE_SynchronInfoData;
	fbExecuteTrigger				 	: r_trig;
	nIndex: uint;
END_VAR

fbExecuteTrigger(clk:=bExecute);
IF fbExecuteTrigger.q THEN
	nStep:=StartSend_MotorParameter_1;
	bBusy:=TRUE;
END_IF

CASE nStep OF
	init:
		bBusy := FALSE;
		bError:=fbWriteCoEParameterEx.bError;
		nErrId:=fbWriteCoEParameterEx.nErrId;
	
	StartSend_MotorParameter_1:
		fbWriteCoEParameterEx(bExecute:=FALSE);
		IF NOT fbWriteCoEParameterEx.bBusy THEN
			TransferStructDataToBuffer_Motor(nChannel:=1);
			fbWriteCoEParameterEx(
				sNetId:= sNetId, 
				nSlaveAddr:= nSlaveAddr, 
				nIndex:= 16#8020, 
				pSrcBuf:= ADR(stCoe_Write_Motor), 
				cbBufLen:= SIZEOF(stCoe_Write_Motor), 
				bExecute:= TRUE,
				bCompleteAccess:= TRUE);
			nStep:=	Sending_MotorParameter_1;
		END_IF

		
	Sending_MotorParameter_1:
		fbWriteCoEParameterEx(bExecute:=FALSE);
		IF NOT fbWriteCoEParameterEx.bBusy THEN
			IF fbWriteCoEParameterEx.bError THEN
				nStep:= init;
			ELSE
				nStep:= StartSend_ControllerParameter_1;
			END_IF
		END_IF
	
	StartSend_ControllerParameter_1:
		fbWriteCoEParameterEx(bExecute:=FALSE);
		IF NOT fbWriteCoEParameterEx.bBusy THEN
			TransferStructDataToBuffer_Controller(nChannel:=1);
			fbWriteCoEParameterEx(
				sNetId:= sNetId, 
				nSlaveAddr:= nSlaveAddr, 
				nIndex:= 16#8023, 
				pSrcBuf:= ADR(stCoe_Write_Controller), 
				cbBufLen:= SIZEOF(stCoe_Write_Controller), 
				bExecute:= TRUE,
				bCompleteAccess:= TRUE);
			nStep:=	Sending_ControllerParameter_1;
		END_IF
		
	Sending_ControllerParameter_1:
		fbWriteCoEParameterEx(bExecute:=FALSE);
		IF NOT fbWriteCoEParameterEx.bBusy THEN
			IF fbWriteCoEParameterEx.bError THEN
				nStep:= init;
			ELSE
				nStep:= StartSend_SynchronInfoData_1;
			END_IF
		END_IF
		
	StartSend_SynchronInfoData_1:		
		fbWriteCoEParameterEx(bExecute:=FALSE);
		IF NOT fbWriteCoEParameterEx.bBusy THEN
			TransferStructDataToBuffer_SynchronInfoData(nChannel:=1);
			fbWriteCoEParameterEx(
				sNetId:= sNetId, 
				nSlaveAddr:= nSlaveAddr, 
				nIndex:= 16#8022, 
				pSrcBuf:= ADR(stCoe_Write_SynchronInfoData), 
				cbBufLen:= SIZEOF(stCoe_Write_SynchronInfoData), 
				bExecute:= TRUE,
				bCompleteAccess:= TRUE);
			nStep:=	Sending_SynchronInfoData_1;
		END_IF
		
	Sending_SynchronInfoData_1:
		fbWriteCoEParameterEx(bExecute:=FALSE);
		IF NOT fbWriteCoEParameterEx.bBusy THEN
			IF fbWriteCoEParameterEx.bError THEN
				nStep:= init;
			ELSE
				nStep:= StartSend_MotorParameter_2;
			END_IF
		END_IF
		
	StartSend_MotorParameter_2:
		fbWriteCoEParameterEx(bExecute:=FALSE);
		IF NOT fbWriteCoEParameterEx.bBusy THEN						
			TransferStructDataToBuffer_Motor(nChannel:=2);
			fbWriteCoEParameterEx(
				sNetId:= sNetId, 
				nSlaveAddr:= nSlaveAddr, 
				nIndex:= 16#8030, 
				pSrcBuf:= ADR(stCoe_Write_Motor), 
				cbBufLen:= SIZEOF(stCoe_Write_Motor), 
				bExecute:= TRUE,
				bCompleteAccess:= TRUE);
			nStep:=	Sending_MotorParameter_2;
		END_IF
		
	Sending_MotorParameter_2:
		fbWriteCoEParameterEx(bExecute:=FALSE);
		IF NOT fbWriteCoEParameterEx.bBusy THEN
			IF fbWriteCoEParameterEx.bError THEN
				nStep:= init;
			ELSE
				nStep:= StartSend_ControllerParameter_2;
			END_IF
		END_IF
	
	StartSend_ControllerParameter_2:
		fbWriteCoEParameterEx(bExecute:=FALSE);
		IF NOT fbWriteCoEParameterEx.bBusy THEN					
			TransferStructDataToBuffer_Controller(nChannel:=2);
			fbWriteCoEParameterEx(
				sNetId:= sNetId, 
				nSlaveAddr:= nSlaveAddr, 
				nIndex:= 16#8033, 
				pSrcBuf:= ADR(stCoe_Write_Controller), 
				cbBufLen:= SIZEOF(stCoe_Write_Controller), 
				bExecute:= TRUE,
				bCompleteAccess:= TRUE);
			nStep:=	Sending_ControllerParameter_2;
		END_IF
		
	Sending_ControllerParameter_2:
		fbWriteCoEParameterEx(bExecute:=FALSE);
		IF NOT fbWriteCoEParameterEx.bBusy THEN
			IF fbWriteCoEParameterEx.bError THEN
				nStep:= init;
			ELSE
				nStep:= StartSend_SynchronInfoData_2;
			END_IF
		END_IF
		
	StartSend_SynchronInfoData_2:
		fbWriteCoEParameterEx(bExecute:=FALSE);
		IF NOT fbWriteCoEParameterEx.bBusy THEN
			TransferStructDataToBuffer_SynchronInfoData(nChannel:=2);
			fbWriteCoEParameterEx(
				sNetId:= sNetId, 
				nSlaveAddr:= nSlaveAddr, 
				nIndex:= 16#8032, 
				pSrcBuf:= ADR(stCoe_Write_SynchronInfoData), 
				cbBufLen:= SIZEOF(stCoe_Write_SynchronInfoData), 
				bExecute:= TRUE,
				bCompleteAccess:= TRUE);
			nStep :=	Sending_SynchronInfoData_2;
		END_IF
		
	Sending_SynchronInfoData_2:
		fbWriteCoEParameterEx(bExecute:=FALSE);
		IF NOT fbWriteCoEParameterEx.bBusy THEN
				nStep:= init;
		END_IF
		
END_CASE

METHOD TransferStructDataToBuffer_Controller
VAR_INPUT
	nChannel:USINT;
END_VAR
// The warning can be disabled here as the user is aware of the risk that the reference may not be valid by checking its validity
{warning disable C0371}
IF nChannel=1 OR nChannel=2 AND __ISVALIDREF(stEP7402_CoE_Parameter) THEN
	stCoe_Write_Controller.Sub_Index_003	:= stEP7402_CoE_Parameter.astCoE_Parameter_Controller[nChannel][E_EP7402_CoE_Controller.Disable_Motor_Diagnosis].nValue.0;            
	stCoe_Write_Controller.Sub_Index_004	:= stEP7402_CoE_Parameter.astCoE_Parameter_Controller[nChannel][E_EP7402_CoE_Controller.Disable_I2T_Current_Limiting].nValue.0;        
	stCoe_Write_Controller.Sub_Index_017	:= stEP7402_CoE_Parameter.astCoE_Parameter_Controller[nChannel][E_EP7402_CoE_Controller.Velocity_Loop_Integral_Time].nValue;         
	stCoe_Write_Controller.Sub_Index_018	:= stEP7402_CoE_Parameter.astCoE_Parameter_Controller[nChannel][E_EP7402_CoE_Controller.Velocity_Loop_Proportional_Gain].nValue;      
	stCoe_Write_Controller.Sub_Index_019	:= TO_USINT(stEP7402_CoE_Parameter.astCoE_Parameter_Controller[nChannel][E_EP7402_CoE_Controller.Velocity_Feed_Forward_Gain].nValue);          
	stCoe_Write_Controller.Sub_Index_020	:= TO_SINT(stEP7402_CoE_Parameter.astCoE_Parameter_Controller[nChannel][E_EP7402_CoE_Controller.Sensorless_Offset_Scaling].nValue);          
	stCoe_Write_Controller.Sub_Index_021	:= TO_UINT(stEP7402_CoE_Parameter.astCoE_Parameter_Controller[nChannel][E_EP7402_CoE_Controller.Align_Duration].nValue);                   
	stCoe_Write_Controller.Sub_Index_024	:= TO_UINT(stEP7402_CoE_Parameter.astCoE_Parameter_Controller[nChannel][E_EP7402_CoE_Controller.Rampup_Duration].nValue);                  
	stCoe_Write_Controller.Sub_Index_025	:= TO_UINT(stEP7402_CoE_Parameter.astCoE_Parameter_Controller[nChannel][E_EP7402_CoE_Controller.Rampup_Velocity].nValue);                  
	stCoe_Write_Controller.Sub_Index_033	:= TO_UINT(stEP7402_CoE_Parameter.astCoE_Parameter_Controller[nChannel][E_EP7402_CoE_Controller.Rampup_Needed_Switchover_Events].nValue);      
	stCoe_Write_Controller.Sub_Index_034	:= TO_UINT(stEP7402_CoE_Parameter.astCoE_Parameter_Controller[nChannel][E_EP7402_CoE_Controller.Commutation_Threshold].nValue);             
	stCoe_Write_Controller.Sub_Index_035	:= TO_UINT(stEP7402_CoE_Parameter.astCoE_Parameter_Controller[nChannel][E_EP7402_CoE_Controller.Current_Loop_Proportional_Gain].nValue);       
	stCoe_Write_Controller.Sub_Index_036	:= TO_UINT(stEP7402_CoE_Parameter.astCoE_Parameter_Controller[nChannel][E_EP7402_CoE_Controller.Current_Loop_Integral_Time].nValue);          
	stCoe_Write_Controller.Sub_Index_037	:= TO_UINT(stEP7402_CoE_Parameter.astCoE_Parameter_Controller[nChannel][E_EP7402_CoE_Controller.Restart_After_Error_Number_Of_Repetition].nValue);
	stCoe_Write_Controller.Sub_Index_038	:= TO_UINT(stEP7402_CoE_Parameter.astCoE_Parameter_Controller[nChannel][E_EP7402_CoE_Controller.Restart_After_Error_Delay].nValue);          
END_IF
END_METHOD

METHOD TransferStructDataToBuffer_Motor
VAR_INPUT
	nChannel:USINT;
END_VAR
// The warning can be disabled here as the user is aware of the risk that the reference may not be valid by checking its validity
{warning disable C0371}

IF nChannel=1 OR nChannel=2 AND __ISVALIDREF(stEP7402_CoE_Parameter) THEN
	stCoe_Write_Motor.Sub_Index_001	:= TO_UINT(stEP7402_CoE_Parameter.astCoE_Parameter_Motor[nChannel][E_EP7402_CoE_Motor.Peak_Current].nValue);
	stCoe_Write_Motor.Sub_Index_002	:= TO_UINT(stEP7402_CoE_Parameter.astCoE_Parameter_Motor[nChannel][E_EP7402_CoE_Motor.Rated_Current].nValue);
	stCoe_Write_Motor.Sub_Index_003	:= TO_UINT(stEP7402_CoE_Parameter.astCoE_Parameter_Motor[nChannel][E_EP7402_CoE_Motor.Rated_Voltage].nValue);
	stCoe_Write_Motor.Sub_Index_004	:= TO_UINT(stEP7402_CoE_Parameter.astCoE_Parameter_Motor[nChannel][E_EP7402_CoE_Motor.Phase_To_Phase_Resistance].nValue);
	stCoe_Write_Motor.Sub_Index_009	:= TO_UINT(stEP7402_CoE_Parameter.astCoE_Parameter_Motor[nChannel][E_EP7402_CoE_Motor.Start_Velocity].nValue);
	stCoe_Write_Motor.Sub_Index_019	:= TO_UINT(stEP7402_CoE_Parameter.astCoE_Parameter_Motor[nChannel][E_EP7402_CoE_Motor.Mechanical_To_Electrical_Ratio].nValue);
	stCoe_Write_Motor.Sub_Index_020	:= TO_UINT(stEP7402_CoE_Parameter.astCoE_Parameter_Motor[nChannel][E_EP7402_CoE_Motor.Rated_Velocity].nValue);
	stCoe_Write_Motor.Sub_Index_022	:= TO_USINT(stEP7402_CoE_Parameter.astCoE_Parameter_Motor[nChannel][E_EP7402_CoE_Motor.I2T_Warn_Level].nValue);
	stCoe_Write_Motor.Sub_Index_024	:= TO_USINT(stEP7402_CoE_Parameter.astCoE_Parameter_Motor[nChannel][E_EP7402_CoE_Motor.I2T_Error_Level].nValue);
	stCoe_Write_Motor.Sub_Index_025	:= TO_UINT(stEP7402_CoE_Parameter.astCoE_Parameter_Motor[nChannel][E_EP7402_CoE_Motor.Motor_Thermal_Time_Constant].nValue);
END_IF
END_METHOD

METHOD TransferStructDataToBuffer_SynchronInfoData
VAR_INPUT
	nChannel:USINT;
END_VAR
// The warning can be disabled here as the user is aware of the risk that the reference may not be valid by checking its validity
{warning disable C0371}

IF nChannel=1 OR nChannel=2 AND __ISVALIDREF(stEP7402_CoE_Parameter) THEN
	stCoe_Write_SynchronInfoData.nInfoData1	:= TO_USINT(stEP7402_CoE_Parameter.astCoE_Parameter_SynchronInfoData[nChannel][1]);
	stCoe_Write_SynchronInfoData.nInfoData2	:= TO_USINT(stEP7402_CoE_Parameter.astCoE_Parameter_SynchronInfoData[nChannel][2]);
	stCoe_Write_SynchronInfoData.nInfoData3	:= TO_USINT(stEP7402_CoE_Parameter.astCoE_Parameter_SynchronInfoData[nChannel][3]);
END_IF
END_METHOD

END_FUNCTION_BLOCK

// ---- POUs/CoE_Access/FB_EP7402_AutoRequestSteps.TcPOU
FUNCTION_BLOCK FB_EP7402_AutoRequestSteps
VAR CONSTANT
	cnValueChannel_1: UINT:=16#800A;
	cnValueChannel_2: UINT:=16#801A;
END_VAR
VAR_INPUT
	bEnable:BOOL;
	tRequestCycleTime:TIME:= T#250mS;
	sNetId 		: T_AmsNetID;
	nSlaveAddr	: UINT;
	bMotorChannel_1:BOOL:= TRUE;
END_VAR
VAR_OUTPUT
	bBusy:BOOL;
	bError:BOOL;
	nErrId:UDINT;
	aResponse:ARRAY [1..6] OF BYTE;
	nMotorStep_Count :UINT;
END_VAR
VAR
	fbTimer:TON;
	fbWriteCoEParameter	:  FB_EcCoESdoWrite;
	fbReadCoEParameter	:  FB_EcCoESdoRead;
	fbReadCoEParameterEx	:  FB_EcCoESdoReadEx;
	fbRequestProgress	: f_trig;
	nStep:(init, request_command_register, requesting_command_register ,send_request, sending_request, request_progress, requesting_progress, request_error, requesting_error);
	fbExecuteTrigger:r_trig;
	nStatus:USINT;
	aBuffer: array [1..12] of Byte;
	fb_f_EnableTrig: f_trig;
	fb_r_EnableTrig: r_trig;
END_VAR

fbTimer(in:= bEnable AND NOT fbTimer.Q, pt:=tRequestCycleTime);

fb_r_EnableTrig(clk:=bEnable);
fb_f_EnableTrig(clk:=bEnable);
IF fb_f_EnableTrig.q THEN
	nStep:=init;
END_IF


CASE nStep OF
	init:
		bBusy := FALSE;
		IF fb_r_EnableTrig.q THEN
			nMotorStep_Count:=0;
			memset(ADR(aResponse),0,SIZEOF(aResponse));
			nStep:=request_command_register;
		END_IF
	
	request_command_register: // Request seems to be necessesary 
		fbReadCoEParameterEx(bExecute:=FALSE);
		IF NOT fbReadCoEParameterEx.bBusy THEN
			fbReadCoEParameterEx(
				sNetId:= sNetId, 
				nSlaveAddr:= nSlaveAddr, 
				nIndex:= 16#FB00, 
				pDstBuf:= ADR(aBuffer), 
				cbBufLen:= SIZEOF(aBuffer), 
				bExecute:= TRUE,
				bCompleteAccess:= TRUE,
				bError=>bError , 
				nErrId=> nErrId);
			nStep:=	requesting_command_register;
		END_IF

		
	requesting_command_register:
		fbReadCoEParameterEx(bExecute:=FALSE);
		IF NOT fbReadCoEParameterEx.bBusy THEN
			IF fbReadCoEParameterEx.bError THEN
				nStep:= init;
			ELSE
				nStep:= send_request;
			END_IF
		END_IF
		
	send_request:
		fbWriteCoEParameter(bExecute:=FALSE);
		IF NOT fbWriteCoEParameter.bBusy AND fbTimer.q THEN
			fbWriteCoEParameter(
				sNetId:= sNetId, 
				nSlaveAddr:=nSlaveAddr , 
				nSubIndex:= 16#1, 
				nIndex:= 16#FB00, 
				pSrcBuf:= SEL(bMotorChannel_1, ADR(cnValueChannel_2), ADR(cnValueChannel_1)), 
				cbBufLen:= SEL(bMotorChannel_1, SIZEOF(cnValueChannel_2), SIZEOF(cnValueChannel_1)),
				bExecute:= TRUE ,
				tTimeout:= ,  
				bError=>bError , 
				nErrId=> nErrId);
			nStep:=	sending_request;
		END_IF

		
	sending_request:
		fbWriteCoEParameter(bExecute:=FALSE);
		IF NOT fbWriteCoEParameter.bBusy THEN
			IF fbWriteCoEParameter.bError THEN
				nStep:= init;
			ELSE
				nStep:= request_progress;
			END_IF
		END_IF
	
	request_progress:
		fbReadCoEParameter(bExecute:=FALSE);
		IF NOT fbReadCoEParameter.bBusy THEN
			fbReadCoEParameter(
				sNetId:= sNetId, 
				nSlaveAddr:= nSlaveAddr, 
				nSubIndex:= 16#2, 
				nIndex:= 16#FB00, 
				pDstBuf:= ADR(nStatus), 
				cbBufLen:= SIZEOF(nStatus), 
				bExecute:= TRUE,
				bError=>bError , 
				nErrId=> nErrId);
			nStep:=	requesting_progress;
		END_IF

		
	requesting_progress:
		fbReadCoEParameter(bExecute:=FALSE);
		IF NOT fbReadCoEParameter.bBusy THEN
			IF fbReadCoEParameter.bError THEN
				nStep:= init;
			ELSE
				IF nStatus=0 THEN
					nStep:= request_command_register;
					nMotorStep_Count:=nMotorStep_Count+1;
				ELSIF nStatus<>0 THEN
					nStep:= request_error;					
				END_IF
			END_IF
		END_IF
		
	request_error:
		fbReadCoEParameter(bExecute:=FALSE);
		IF NOT fbReadCoEParameter.bBusy THEN
			fbReadCoEParameter(
				sNetId:= sNetId, 
				nSlaveAddr:= nSlaveAddr, 
				nSubIndex:= 16#3, 
				nIndex:= 16#FB00, 
				pDstBuf:= ADR(aResponse), 
				cbBufLen:= SIZEOF(aResponse), 
				bExecute:= TRUE,
				bError=> bError , 
				nErrId=> nErrId);
			nStep:=	requesting_error;
		END_IF

		
	requesting_error:
		fbReadCoEParameter(bExecute:=FALSE);
		IF NOT fbReadCoEParameter.bBusy THEN
				nStep:= init;
		END_IF
	
END_CASE

END_FUNCTION_BLOCK

// ---- POUs/CoE_Access/FB_EP7402_Scan_Motor.TcPOU
FUNCTION_BLOCK FB_EP7402_Scan_Motor
VAR CONSTANT
	cnValueChannel_1: UINT:=16#8007;
	cnValueChannel_2: UINT:=16#8017;
END_VAR
VAR_INPUT
	bExecute:BOOL;
	sNetId 		: T_AmsNetID;
	tUpdateInterval:TIME:=T#1S;
	nSlaveAddr	: UINT;
	bMotorChannel_1:BOOL:= TRUE;
END_VAR
VAR_OUTPUT
	bBusy:BOOL;
	nProgress: USINT;
	aResponse:ARRAY [1..6] OF BYTE;
	bError:BOOL;
	nErrId:UDINT;
END_VAR
VAR
	fbWriteCoEParameter	:  FB_EcCoESdoWrite;
	fbReadCoEParameter	:  FB_EcCoESdoRead;
	fbReadCoEParameterEx	:  FB_EcCoESdoReadEx;
	fbRequestProgress:f_trig;
	nStep:(init, request_command_register, requesting_command_register ,send_request, sending_request, request_progress, requesting_progress, request_error, requesting_error);
	fbExecuteTrigger:r_trig;
	nStatus:USINT;
	aBuffer: array [1..12] of Byte;
	
END_VAR

fbExecuteTrigger(clk:=bExecute);
IF fbExecuteTrigger.q THEN
	nStep:=request_command_register;
	nProgress:=0;
	memset(ADR(aResponse),0,SIZEOF(aResponse));
	bBusy:=TRUE;
END_IF



CASE nStep OF
	init:
		bBusy := FALSE;
	
	request_command_register:
		fbReadCoEParameterEx(bExecute:=FALSE);
		IF NOT fbReadCoEParameterEx.bBusy THEN
			fbReadCoEParameterEx(
				sNetId:= sNetId, 
				nSlaveAddr:= nSlaveAddr, 
				nIndex:= 16#FB00, 
				pDstBuf:= ADR(aBuffer), 
				cbBufLen:= SIZEOF(aBuffer), 
				bExecute:= TRUE,
				bCompleteAccess:= TRUE,
				bError=>bError , 
				nErrId=> nErrId);
			nStep:=	requesting_command_register;
		END_IF

		
	requesting_command_register:
		fbReadCoEParameterEx(bExecute:=FALSE);
		IF NOT fbReadCoEParameterEx.bBusy THEN
			IF fbReadCoEParameterEx.bError THEN
				nStep:= init;
			ELSE
				nStep:= send_request;
			END_IF
		END_IF
		
	send_request:
		fbWriteCoEParameter(bExecute:=FALSE);
		IF NOT fbWriteCoEParameter.bBusy THEN
			fbWriteCoEParameter(
				sNetId:= sNetId, 
				nSlaveAddr:=nSlaveAddr , 
				nSubIndex:= 16#1, 
				nIndex:= 16#FB00, 
				pSrcBuf:= SEL(bMotorChannel_1, ADR(cnValueChannel_2), ADR(cnValueChannel_1)), 
				cbBufLen:= SEL(bMotorChannel_1, SIZEOF(cnValueChannel_2), SIZEOF(cnValueChannel_1)),
				bExecute:= TRUE ,
				tTimeout:= ,  
				bError=>bError , 
				nErrId=> nErrId);
			nStep:=	sending_request;
		END_IF

		
	sending_request:
		fbWriteCoEParameter(bExecute:=FALSE);
		IF NOT fbWriteCoEParameter.bBusy THEN
			IF fbWriteCoEParameter.bError THEN
				nStep:= init;
			ELSE
				nStep:= request_progress;
			END_IF
		END_IF
	
	request_progress:
		fbReadCoEParameter(bExecute:=FALSE);
		IF NOT fbReadCoEParameter.bBusy THEN
			fbReadCoEParameter(
				sNetId:= sNetId, 
				nSlaveAddr:= nSlaveAddr, 
				nSubIndex:= 16#2, 
				nIndex:= 16#FB00, 
				pDstBuf:= ADR(nStatus), 
				cbBufLen:= SIZEOF(nStatus), 
				bExecute:= TRUE,
				bError=>bError , 
				nErrId=> nErrId);
			nStep:=	requesting_progress;
		END_IF

		
	requesting_progress:
		fbReadCoEParameter(bExecute:=FALSE);
		IF NOT fbReadCoEParameter.bBusy THEN
			IF fbReadCoEParameter.bError THEN
				nStep:= init;
			ELSE
				IF nStatus>100 THEN
					nProgress:=nStatus-100;
					nStep:= request_progress;
				ELSIF nStatus=0 THEN
					nProgress:=100;
					nStep:= init;
				ELSE
					nProgress:=0;
					nStep:= request_error;					
				END_IF
			END_IF
		END_IF
		
	request_error:
		fbReadCoEParameter(bExecute:=FALSE);
		IF NOT fbReadCoEParameter.bBusy THEN
			fbReadCoEParameter(
				sNetId:= sNetId, 
				nSlaveAddr:= nSlaveAddr, 
				nSubIndex:= 16#3, 
				nIndex:= 16#FB00, 
				pDstBuf:= ADR(aResponse), 
				cbBufLen:= SIZEOF(aResponse), 
				bExecute:= TRUE,
				bError=> bError , 
				nErrId=> nErrId);
			nStep:=	requesting_error;
		END_IF

		
	requesting_error:
		fbReadCoEParameter(bExecute:=FALSE);
		IF NOT fbReadCoEParameter.bBusy THEN
				nStep:= init;
		END_IF
	
END_CASE

END_FUNCTION_BLOCK
